PROGRAM P_MachineControl
VAR
	fbManualControlWinch 		: FB_ManualControl;
	fbManualControlCyl	 		: FB_ManualControl;
	//fbAutomaticControlWinch 	: FB_AutomaticControl_old;
	//fbAutomaticControlCyl	 	: FB_AutomaticControl_old;
	fWinchControlSignalManual 			: LREAL;
	fCylControlSignalManual 			: LREAL;
	fWinchControlSignalAuto 			: LREAL;
	fCylControlSignalAuto				: LREAL;
	fbAutomaticControlWinch 	:	FB_AutomaticControl;
	fbAutomaticControlCylinder 		:	FB_AutomaticControl;
	fbModifyAutomaticControlSettingsWinch : FB_ModifyAutomaticControlSettings;
	fbModifyAutomaticControlSettingsCylinder : FB_ModifyAutomaticControlSettings;
END_VAR

G_Work.bManualMode := G_Inputs.bManualModeSelector;
G_Work.bAutoMode := G_Inputs.bAutoModeSelector;

G_Work.bWinchEnable := (G_Hmi.bWinchEnable AND G_Inputs.bJoystickEnable);
G_Work.bCylEnable :=  (G_Hmi.bCylEnable AND G_Inputs.bJoystickEnable);

fbManualControlWinch(
	bEnable := G_Work.bManualMode AND G_Work.bWinchEnable,
	fInput := G_Sensors.fJoystickNormalizedY*-G_Parameters.stParam.fWinchSpeedReducerGain,
	fControlRefSignal => fWinchControlSignalManual
);

fbManualControlCyl(
	bEnable := G_Work.bManualMode AND G_Work.bCylEnable,
	fInput := G_Sensors.fJoystickNormalizedX*G_Parameters.stParam.fCylSpeedReducerGain,
	fControlRefSignal => fCylControlSignalManual
);

//fbAutomaticControlWinch(
//	bEnable := G_Work.bAutoMode AND G_Hmi.bWinchEnable,
//	bStartMotion := G_Inputs.bStartButton,
//	bStopMotion := G_Inputs.bStopButton,
//	stValveOutputGeneratorSettings := G_Parameters.stWinchValveOutputGeneratorSettings,
//	fNormalizedValveOpeningRefSignal => fWinchControlSignalAuto,
//	fTime => G_Work.fWinchTime
//);

//fbAutomaticControlCyl(
//	bEnable := G_Work.bAutoMode AND G_Hmi.bCylEnable,
//	bStartMotion := G_Inputs.bStartButton,
//	bStopMotion := G_Inputs.bStopButton,
//	stValveOutputGeneratorSettings := G_Parameters.stCylValveOutputGeneratorSettings,
//	fNormalizedValveOpeningRefSignal => fCylControlSignalAuto,
//	fTime => G_Work.fCylTime
//);

fbModifyAutomaticControlSettingsWinch(
	stParamOpenLoopControllSettings := G_Parameters.stParam.stOpenLoopControlSettingsWinch,
	stParamClosedLoopControllSettings := G_Parameters.stParam.stClosedLoopControlSettingsWinch,	
	stModify := G_Hmi.stModifyAutomaticControlSettingsWinch
);

fbAutomaticControlWinch(
	bEnable := G_Work.bAutoMode AND G_Hmi.bWinchEnable,
	bStartMotion := G_Inputs.bStartButton,
	bStopMotion := G_Inputs.bStopButton,
	stMotionReferenceGeneratorSettings := G_Hmi.stMotionReferenceGeneratorSettingsWinch,
	stAutomaticControlSettings := G_Hmi.stAutomaticControlSettingsWinch,
	stClosedLoopControlSettings := G_Parameters.stParam.stClosedLoopControlSettingsWinch,
	stOpenLoopControlSettings := G_Parameters.stParam.stOpenLoopControlSettingsWinch,
	stParam := G_Parameters.stParam,
	fPositionFeedback := G_Sensors.fWinchWirePosition,
	fVelocityReference_ms => G_Work.fVelRefWinch,
	fPositionReference_m => G_Work.fPosRefWinch,
	fTime => G_Work.fWinchTime,
	fPositionError_mm => G_Work.fPositionErrorWinch_mm,
	fControlOutputNormalized => G_Work.fControlSignWinch
);


fbModifyAutomaticControlSettingsCylinder(
	stParamOpenLoopControllSettings := G_Parameters.stParam.stOpenLoopControlSettingsCylinder,
	stParamClosedLoopControllSettings := G_Parameters.stParam.stClosedLoopControlSettingsCylinder,	
	stModify := G_Hmi.stModifyAutomaticControlSettingsCylinder
);

fbAutomaticControlCylinder(
	bEnable := G_Work.bAutoMode AND G_Hmi.bCylEnable,
	bStartMotion := G_Inputs.bStartButton,
	bStopMotion := G_Inputs.bStopButton,
	stMotionReferenceGeneratorSettings := G_Hmi.stMotionReferenceGeneratorSettingsCylinder,
	stAutomaticControlSettings := G_Hmi.stAutomaticControlSettingsCylinder,
	stClosedLoopControlSettings := G_Parameters.stParam.stClosedLoopControlSettingsCylinder,
	stOpenLoopControlSettings := G_Parameters.stParam.stOpenLoopControlSettingsCylinder,
	stParam := G_Parameters.stParam,
	fPositionFeedback := G_Sensors.fPositionCylPiston,
	fVelocityReference_ms => G_Work.fVelRefCyl,
	fPositionReference_m => G_Work.fPosRefCyl,
	fTime => G_Work.fCylTime,
	fPositionError_mm => G_Work.fPositionErrorCylinder_mm,
	fControlOutputNormalized => G_Work.fControlSignCyl
);

IF G_Work.bManualMode THEN
	G_Work.fWinchControlInput := fWinchControlSignalManual;
	G_Work.fCylControlInput := fCylControlSignalManual;
ELSIF G_Work.bAutoMode THEN
	G_Work.fWinchControlInput := G_Work.fControlSignWinch;
	G_Work.fCylControlInput := -G_Work.fControlSignCyl;
ELSE
	G_Work.fWinchControlInput := 0.0; 
	G_Work.fCylControlInput := 0.0;
END_IF

END_PROGRAM

(* stored: Version 1.1.0.1, ProductVersion 3.1.4024.11
   POU P_MachineControl: Id {a90e0789-57c0-407b-b2f1-afc96a165b42}, SpecialFunc None *)
